// TIA Portal V19 export
TYPE "Positioning_EPOS_Machine_Alr"
// stored: Access Published
   STRUCT
      S120_Fault : Bool;   // Fault message(s) in the SINAMICS drive
      S120_ComErr : Bool;   // Interruption of communication to the SINAMICS drive
      S120_WriteParErr : Bool;   // SinaPara wirte par error
      Ax_NotHomed : Bool;   // Axis is NOT homed / refereced
      Ax_ErrSelMode : Bool;   // Incorrect operating mode selected
      Ax_ErrOverride : Bool;   // Incorrect parameterization of the override inputs
      Ax_InvalidTraversingBlockNr : Bool;   // Invalid traversing block number
      HwLimitMinus : Bool;   // Negative limit switch reached / exceeded
      HwLimitPlus : Bool;   // Positive limit switch reached / exceeded
      BrakeTimeOut : Bool;   // Brake feedback timeout
      Fan_M : "MotorAlr";   // MOTOR FAN
   END_STRUCT;
END_TYPE
